LIN {X 0,Y 105.702,Z 1204.492,A -85,B 0,C 180,E1 2560.823,E2 2560.823} C_VEL
LIN {X 0,Y 120.882,Z 1198.363,A -85,B 0,C 180,E1 2552.47,E2 2552.47} C_VEL
LIN {X 0,Y 137.979,Z 1190.359,A -85,B 0,C 180,E1 2546.031,E2 2546.031} C_VEL
LIN {X 0,Y 156.407,Z 1180.629,A -85,B 0,C 180,E1 2541.04,E2 2541.04} C_VEL
LIN {X 0,Y 173.081,Z 1170.511,A -85,B 0,C 180,E1 2537.603,E2 2537.603} C_VEL
LIN {X 0,Y 192.101,Z 1157.421,A -85,B 0,C 180,E1 2534.511,E2 2534.511} C_VEL
LIN {X 0,Y 207.848,Z 1145.066,A -85,B 0,C 180,E1 2532.437,E2 2532.437} C_VEL
LIN {X 0,Y 225.86,Z 1129.001,A -85,B 0,C 180,E1 2530.458,E2 2530.458} C_VEL
LIN {X 0,Y 241.449,Z 1113.168,A -85,B 0,C 180,E1 2529.016,E2 2529.016} C_VEL
LIN {X 0,Y 256.349,Z 1095.766,A -85,B 0,C 180,E1 2527.823,E2 2527.823} C_VEL
LIN {X 0,Y 270.386,Z 1077.144,A -85,B 0,C 180,E1 2526.842,E2 2526.842} C_VEL
LIN {X 0,Y 283.038,Z 1057.453,A -85,B 0,C 180,E1 2526.055,E2 2526.055} C_VEL
LIN {X 0,Y 294.767,Z 1036.226,A -85,B 0,C 180,E1 2525.403,E2 2525.403} C_VEL
LIN {X 0,Y 304.085,Z 1016.178,A -85,B 0,C 180,E1 2524.939,E2 2524.939} C_VEL
LIN {X 0,Y 312.937,Z 993.046,A -85,B 0,C 180,E1 2524.54,E2 2524.54} C_VEL
LIN {X 0,Y 319.741,Z 970.772,A -85,B 0,C 180,E1 2524.255,E2 2524.255} C_VEL
LIN {X 0,Y 324.96,Z 947.508,A -85,B 0,C 180,E1 2523.991,E2 2523.991} C_VEL
LIN {X 0,Y 328.847,Z 922.27,A -85,B 0,C 180,E1 2523.717,E2 2523.717} C_VEL
LIN {X 0,Y 337.296,Z 853.105,A -85,B 0,C 180,E1 2522.984,E2 2522.984} C_VEL
LIN {X 0,Y 326.597,Z 938.266,A -85,B 0,C 180,E1 2522.039,E2 2522.039} C_VEL
LIN {X 0,Y 321.884,Z 961.652,A -85,B 0,C 180,E1 2521.748,E2 2521.748} C_VEL
LIN {X 0,Y 315.799,Z 984.104,A -85,B 0,C 180,E1 2521.402,E2 2521.402} C_VEL
LIN {X 0,Y 307.999,Z 1006.102,A -85,B 0,C 180,E1 2520.96,E2 2520.96} C_VEL
LIN {X 0,Y 298.407,Z 1028.316,A -85,B 0,C 180,E1 2520.384,E2 2520.384} C_VEL
LIN {X 0,Y 288.461,Z 1047.548,A -85,B 0,C 180,E1 2519.758,E2 2519.758} C_VEL
LIN {X 0,Y 275.512,Z 1068.916,A -85,B 0,C 180,E1 2518.888,E2 2518.888} C_VEL
LIN {X 0,Y 262.518,Z 1087.397,A -85,B 0,C 180,E1 2517.935,E2 2517.935} C_VEL
LIN {X 0,Y 247.376,Z 1106.017,A -85,B 0,C 180,E1 2516.694,E2 2516.694} C_VEL
LIN {X 0,Y 231.767,Z 1122.947,A -85,B 0,C 180,E1 2515.238,E2 2515.238} C_VEL
LIN {X 0,Y 215.365,Z 1138.404,A -85,B 0,C 180,E1 2513.473,E2 2513.473} C_VEL
LIN {X 0,Y 197.315,Z 1153.508,A -85,B 0,C 180,E1 2511.16,E2 2511.16} C_VEL
LIN {X 0,Y 179.971,Z 1166.226,A -85,B 0,C 180,E1 2508.462,E2 2508.462} C_VEL
LIN {X 0,Y 175.041,Z 1169.634,A -85,B 0,C 180,E1 2507.581,E2 2507.581} C_VEL
LIN {X 0,Y 168.74,Z 1173.521,A -85,B 0,C 180,E1 2506.765,E2 2506.765} C_VEL
LIN {X 0,Y 150.312,Z 1183.482,A -85,B 0,C 180,E1 2505.451,E2 2505.451} C_VEL
LIN {X 0,Y 144.844,Z 1186.245,A -85,B 0,C 180,E1 2504.485,E2 2504.485} C_VEL
LIN {X 0,Y 126.307,Z 1195.602,A -85,B 0,C 180,E1 2499.083,E2 2499.083} C_VEL
LIN {X 0,Y 108.864,Z 1203.189,A -85,B 0,C 180,E1 2491.849,E2 2491.849} C_VEL
LIN {X 0,Y 93.007,Z 1209.46,A -85,B 0,C 180,E1 2481.7,E2 2481.7} C_VEL
LIN {X 0,Y 81.228,Z 1213.752,A -85,B 0,C 180,E1 2468.886,E2 2468.886} C_VEL
LIN {X 0,Y 73.84,Z 1216.677,A -85,B 0,C 180,E1 2452.281,E2 2452.281} C_VEL
LIN {X 0,Y 72.017,Z 1217.75,A -85,B 0,C 180,E1 2437.98,E2 2437.98} C_VEL
LIN {X 0,Y 72.03,Z 1217.944,A -85,B 0,C 180,E1 2428.409,E2 2428.409} C_VEL
LIN {X 0,Y 72.337,Z 1217.462,A -85,B 0,C 180,E1 2416.41,E2 2416.41} C_VEL
LIN {X 0,Y 76.053,Z 1215.666,A -85,B 0,C 180,E1 2400.894,E2 2400.894} C_VEL
LIN {X 0,Y 85.042,Z 1212.358,A -85,B 0,C 180,E1 2386.078,E2 2386.078} C_VEL
LIN {X 0,Y 98.855,Z 1207.101,A -85,B 0,C 180,E1 2373.965,E2 2373.965} C_VEL
LIN {X 0,Y 115.778,Z 1200.203,A -85,B 0,C 180,E1 2364.936,E2 2364.936} C_VEL
LIN {X 0,Y 133.031,Z 1192.152,A -85,B 0,C 180,E1 2358.736,E2 2358.736} C_VEL
LIN {X 0,Y 152.349,Z 1181.996,A -85,B 0,C 180,E1 2353.757,E2 2353.757} C_VEL
LIN {X 0,Y 169.742,Z 1171.523,A -85,B 0,C 180,E1 2350.358,E2 2350.358} C_VEL
LIN {X 0,Y 189.984,Z 1157.647,A -85,B 0,C 180,E1 2347.257,E2 2347.257} C_VEL
LIN {X 0,Y 207.781,Z 1143.722,A -85,B 0,C 180,E1 2345.065,E2 2345.065} C_VEL
LIN {X 0,Y 225.332,Z 1127.955,A -85,B 0,C 180,E1 2343.257,E2 2343.257} C_VEL
LIN {X 0,Y 241.589,Z 1111.448,A -85,B 0,C 180,E1 2341.832,E2 2341.832} C_VEL
LIN {X 0,Y 256.663,Z 1093.76,A -85,B 0,C 180,E1 2340.67,E2 2340.67} C_VEL
LIN {X 0,Y 271.466,Z 1073.856,A -85,B 0,C 180,E1 2339.652,E2 2339.652} C_VEL
LIN {X 0,Y 283.511,Z 1055.087,A -85,B 0,C 180,E1 2338.901,E2 2338.901} C_VEL
LIN {X 0,Y 295.099,Z 1033.92,A -85,B 0,C 180,E1 2338.225,E2 2338.225} C_VEL
LIN {X 0,Y 304.701,Z 1013.197,A -85,B 0,C 180,E1 2337.702,E2 2337.702} C_VEL
LIN {X 0,Y 312.808,Z 991.691,A -85,B 0,C 180,E1 2337.278,E2 2337.278} C_VEL
LIN {X 0,Y 317.419,Z 977.052,A -85,B 0,C 180,E1 2337.025,E2 2337.025} C_VEL
LIN {X 0,Y 309.956,Z 999.939,A -85,B 0,C 180,E1 2336.744,E2 2336.744} C_VEL
LIN {X 0,Y 301.552,Z 1020.488,A -85,B 0,C 180,E1 2336.4,E2 2336.4} C_VEL
LIN {X 0,Y 290.701,Z 1042.634,A -85,B 0,C 180,E1 2335.902,E2 2335.902} C_VEL
LIN {X 0,Y 279.88,Z 1061.31,A -85,B 0,C 180,E1 2335.352,E2 2335.352} C_VEL
LIN {X 0,Y 266.156,Z 1081.659,A -85,B 0,C 180,E1 2334.57,E2 2334.57} C_VEL
LIN {X 0,Y 252.01,Z 1099.859,A -85,B 0,C 180,E1 2333.65,E2 2333.65} C_VEL
LIN {X 0,Y 236.489,Z 1117.088,A -85,B 0,C 180,E1 2332.5,E2 2332.5} C_VEL
LIN {X 0,Y 220.612,Z 1132.702,A -85,B 0,C 180,E1 2331.121,E2 2331.121} C_VEL
LIN {X 0,Y 203.466,Z 1147.304,A -85,B 0,C 180,E1 2329.365,E2 2329.365} C_VEL
LIN {X 0,Y 184.695,Z 1161.384,A -85,B 0,C 180,E1 2327.018,E2 2327.018} C_VEL
LIN {X 0,Y 167.217,Z 1172.785,A -85,B 0,C 180,E1 2324.298,E2 2324.298} C_VEL
LIN {X 0,Y 147.575,Z 1183.95,A -85,B 0,C 180,E1 2320.349,E2 2320.349} C_VEL
LIN {X 0,Y 129.663,Z 1192.8,A -85,B 0,C 180,E1 2315.494,E2 2315.494} C_VEL
LIN {X 0,Y 111.422,Z 1200.526,A -85,B 0,C 180,E1 2308.484,E2 2308.484} C_VEL
LIN {X 0,Y 95.371,Z 1206.516,A -85,B 0,C 180,E1 2299.011,E2 2299.011} C_VEL
LIN {X 0,Y 83.103,Z 1210.53,A -85,B 0,C 180,E1 2286.983,E2 2286.983} C_VEL
LIN {X 0,Y 74.655,Z 1213.263,A -85,B 0,C 180,E1 2270.357,E2 2270.357} C_VEL
LIN {X 0,Y 72.2,Z 1214.155,A -85,B 0,C 180,E1 2255.563,E2 2255.563} C_VEL
LIN {X 0,Y 72.16,Z 1214.185,A -85,B 0,C 180,E1 2245.231,E2 2245.231} C_VEL
LIN {X 0,Y 74,Z 1213.483,A -85,B 0,C 180,E1 2231.895,E2 2231.895} C_VEL
LIN {X 0,Y 80.832,Z 1211.371,A -85,B 0,C 180,E1 2216.177,E2 2216.177} C_VEL
LIN {X 0,Y 92.82,Z 1207.406,A -85,B 0,C 180,E1 2202.904,E2 2202.904} C_VEL
LIN {X 0,Y 109.122,Z 1201.539,A -85,B 0,C 180,E1 2192.545,E2 2192.545} C_VEL
LIN {X 0,Y 125.492,Z 1194.778,A -85,B 0,C 180,E1 2185.799,E2 2185.799} C_VEL
LIN {X 0,Y 144.029,Z 1185.943,A -85,B 0,C 180,E1 2180.417,E2 2180.417} C_VEL
LIN {X 0,Y 161.73,Z 1176.279,A -85,B 0,C 180,E1 2176.615,E2 2176.615} C_VEL
LIN {X 0,Y 180.001,Z 1164.784,A -85,B 0,C 180,E1 2173.572,E2 2173.572} C_VEL
LIN {X 0,Y 197.751,Z 1152.12,A -85,B 0,C 180,E1 2171.22,E2 2171.22} C_VEL
LIN {X 0,Y 214.827,Z 1138.084,A -85,B 0,C 180,E1 2169.357,E2 2169.357} C_VEL
LIN {X 0,Y 231.141,Z 1122.991,A -85,B 0,C 180,E1 2167.865,E2 2167.865} C_VEL
LIN {X 0,Y 246.625,Z 1106.46,A -85,B 0,C 180,E1 2166.652,E2 2166.652} C_VEL
LIN {X 0,Y 261.237,Z 1088.836,A -85,B 0,C 180,E1 2165.662,E2 2165.662} C_VEL
LIN {X 0,Y 274.451,Z 1070.287,A -85,B 0,C 180,E1 2164.87,E2 2164.87} C_VEL
LIN {X 0,Y 287.221,Z 1049.628,A -85,B 0,C 180,E1 2164.192,E2 2164.192} C_VEL
LIN {X 0,Y 297.576,Z 1029.866,A -85,B 0,C 180,E1 2163.697,E2 2163.697} C_VEL
LIN {X 0,Y 307.457,Z 1007.353,A -85,B 0,C 180,E1 2163.274,E2 2163.274} C_VEL
LIN {X 0,Y 315.059,Z 986.183,A -85,B 0,C 180,E1 2162.986,E2 2162.986} C_VEL
LIN {X 0,Y 316.8,Z 980.517,A -85,B 0,C 180,E1 2162.918,E2 2162.918} C_VEL
LIN {X 0,Y 308.808,Z 1003.784,A -85,B 0,C 180,E1 2162.503,E2 2162.503} C_VEL
LIN {X 0,Y 300.145,Z 1024.367,A -85,B 0,C 180,E1 2162.032,E2 2162.032} C_VEL
LIN {X 0,Y 289.549,Z 1045.161,A -85,B 0,C 180,E1 2161.44,E2 2161.44} C_VEL
LIN {X 0,Y 277.655,Z 1065.235,A -85,B 0,C 180,E1 2160.725,E2 2160.725} C_VEL
LIN {X 0,Y 264.462,Z 1084.134,A -85,B 0,C 180,E1 2159.872,E2 2159.872} C_VEL
LIN {X 0,Y 249.52,Z 1102.865,A -85,B 0,C 180,E1 2158.787,E2 2158.787} C_VEL
LIN {X 0,Y 234.183,Z 1119.573,A -85,B 0,C 180,E1 2157.535,E2 2157.535} C_VEL
LIN {X 0,Y 216.533,Z 1136.41,A -85,B 0,C 180,E1 2155.863,E2 2155.863} C_VEL
LIN {X 0,Y 199.097,Z 1151.041,A -85,B 0,C 180,E1 2153.905,E2 2153.905} C_VEL
LIN {X 0,Y 180.729,Z 1164.455,A -85,B 0,C 180,E1 2151.409,E2 2151.409} C_VEL
LIN {X 0,Y 162.233,Z 1176.458,A -85,B 0,C 180,E1 2148.265,E2 2148.265} C_VEL
LIN {X 0,Y 144.844,Z 1186.245,A -85,B 0,C 180,E1 2144.485,E2 2144.485} C_VEL
LIN {X 0,Y 138.393,Z 1189.511,A -85,B 0,C 180,E1 2143.29,E2 2143.29} C_VEL
LIN {X 0,Y 120.351,Z 1196.925,A -85,B 0,C 180,E1 2141.09,E2 2141.09} C_VEL
LIN {X 0,Y 113.904,Z 1199.508,A -85,B 0,C 180,E1 2139.414,E2 2139.414} C_VEL
LIN {X 0,Y 95.954,Z 1206.45,A -85,B 0,C 180,E1 2131.08,E2 2131.08} C_VEL
LIN {X 0,Y 81.07,Z 1211.613,A -85,B 0,C 180,E1 2119.877,E2 2119.877} C_VEL
LIN {X 0,Y 69.737,Z 1215.254,A -85,B 0,C 180,E1 2103.998,E2 2103.998} C_VEL
LIN {X 0,Y 64.714,Z 1217.132,A -85,B 0,C 180,E1 2087.071,E2 2087.071} C_VEL
LIN {X 0,Y 64.013,Z 1217.723,A -85,B 0,C 180,E1 2072.686,E2 2072.686} C_VEL
LIN {X 0,Y 64.003,Z 1217.615,A -85,B 0,C 180,E1 2063.722,E2 2063.722} C_VEL
LIN {X 0,Y 65.464,Z 1216.757,A -85,B 0,C 180,E1 2048.703,E2 2048.703} C_VEL
LIN {X 0,Y 72.619,Z 1214.323,A -85,B 0,C 180,E1 2030.702,E2 2030.702} C_VEL
LIN {X 0,Y 84.806,Z 1210.252,A -85,B 0,C 180,E1 2016.706,E2 2016.706} C_VEL
LIN {X 0,Y 101.269,Z 1204.428,A -85,B 0,C 180,E1 2006.043,E2 2006.043} C_VEL
LIN {X 0,Y 118.415,Z 1197.441,A -85,B 0,C 180,E1 1998.97,E2 1998.97} C_VEL
LIN {X 0,Y 138.672,Z 1188.015,A -85,B 0,C 180,E1 1993.251,E2 1993.251} C_VEL
LIN {X 0,Y 157.115,Z 1178.086,A -85,B 0,C 180,E1 1989.461,E2 1989.461} C_VEL
LIN {X 0,Y 177.052,Z 1165.75,A -85,B 0,C 180,E1 1986.324,E2 1986.324} C_VEL
LIN {X 0,Y 195.455,Z 1152.75,A -85,B 0,C 180,E1 1984.031,E2 1984.031} C_VEL
LIN {X 0,Y 213.903,Z 1137.723,A -85,B 0,C 180,E1 1982.143,E2 1982.143} C_VEL
LIN {X 0,Y 231.481,Z 1121.442,A -85,B 0,C 180,E1 1980.634,E2 1980.634} C_VEL
LIN {X 0,Y 246.974,Z 1104.919,A -85,B 0,C 180,E1 1979.483,E2 1979.483} C_VEL
LIN {X 0,Y 263.061,Z 1085.24,A -85,B 0,C 180,E1 1978.43,E2 1978.43} C_VEL
LIN {X 0,Y 276.189,Z 1066.705,A -85,B 0,C 180,E1 1977.666,E2 1977.666} C_VEL
LIN {X 0,Y 284.295,Z 1053.752,A -85,B 0,C 180,E1 1977.214,E2 1977.214} C_VEL
LIN {X 0,Y 271.987,Z 1072.972,A -85,B 0,C 180,E1 1976.628,E2 1976.628} C_VEL
LIN {X 0,Y 256.654,Z 1093.584,A -85,B 0,C 180,E1 1975.794,E2 1975.794} C_VEL
LIN {X 0,Y 241.933,Z 1110.756,A -85,B 0,C 180,E1 1974.874,E2 1974.874} C_VEL
LIN {X 0,Y 225.34,Z 1127.498,A -85,B 0,C 180,E1 1973.674,E2 1973.674} C_VEL
LIN {X 0,Y 207.908,Z 1142.981,A -85,B 0,C 180,E1 1972.172,E2 1972.172} C_VEL
LIN {X 0,Y 190.648,Z 1156.247,A -85,B 0,C 180,E1 1970.391,E2 1970.391} C_VEL
LIN {X 0,Y 171.743,Z 1169.043,A -85,B 0,C 180,E1 1967.977,E2 1967.977} C_VEL
LIN {X 0,Y 153.222,Z 1179.86,A -85,B 0,C 180,E1 1964.968,E2 1964.968} C_VEL
LIN {X 0,Y 132.596,Z 1190.229,A -85,B 0,C 180,E1 1960.489,E2 1960.489} C_VEL
LIN {X 0,Y 113.874,Z 1198.315,A -85,B 0,C 180,E1 1954.74,E2 1954.74} C_VEL
LIN {X 0,Y 95.933,Z 1204.811,A -85,B 0,C 180,E1 1946.49,E2 1946.49} C_VEL
LIN {X 0,Y 80.678,Z 1209.653,A -85,B 0,C 180,E1 1934.944,E2 1934.944} C_VEL
LIN {X 0,Y 70.026,Z 1212.639,A -85,B 0,C 180,E1 1919.983,E2 1919.983} C_VEL
LIN {X 0,Y 64.708,Z 1214.235,A -85,B 0,C 180,E1 1901.588,E2 1901.588} C_VEL
LIN {X 0,Y 64.092,Z 1214.476,A -85,B 0,C 180,E1 1888.212,E2 1888.212} C_VEL
LIN {X 0,Y 65.755,Z 1213.882,A -85,B 0,C 180,E1 1872.295,E2 1872.295} C_VEL
LIN {X 0,Y 71.984,Z 1212.139,A -85,B 0,C 180,E1 1856.248,E2 1856.248} C_VEL
LIN {X 0,Y 84.9,Z 1208.419,A -85,B 0,C 180,E1 1841.086,E2 1841.086} C_VEL
LIN {X 0,Y 100.349,Z 1203.42,A -85,B 0,C 180,E1 1831.032,E2 1831.032} C_VEL
LIN {X 0,Y 118.798,Z 1196.378,A -85,B 0,C 180,E1 1823.453,E2 1823.453} C_VEL
LIN {X 0,Y 137.838,Z 1187.977,A -85,B 0,C 180,E1 1818.148,E2 1818.148} C_VEL
LIN {X 0,Y 156.838,Z 1178.026,A -85,B 0,C 180,E1 1814.301,E2 1814.301} C_VEL
LIN {X 0,Y 176.392,Z 1166.281,A -85,B 0,C 180,E1 1811.296,E2 1811.296} C_VEL
LIN {X 0,Y 193.469,Z 1154.447,A -85,B 0,C 180,E1 1809.215,E2 1809.215} C_VEL
LIN {X 0,Y 213.018,Z 1138.919,A -85,B 0,C 180,E1 1807.281,E2 1807.281} C_VEL
LIN {X 0,Y 229.203,Z 1124.197,A -85,B 0,C 180,E1 1805.953,E2 1805.953} C_VEL
LIN {X 0,Y 245.334,Z 1107.345,A -85,B 0,C 180,E1 1804.824,E2 1804.824} C_VEL
LIN {X 0,Y 260.076,Z 1089.844,A -85,B 0,C 180,E1 1803.936,E2 1803.936} C_VEL
LIN {X 0,Y 273.888,Z 1070.725,A -85,B 0,C 180,E1 1803.202,E2 1803.202} C_VEL
LIN {X 0,Y 283.669,Z 1055.389,A -85,B 0,C 180,E1 1802.726,E2 1802.726} C_VEL
LIN {X 0,Y 271.636,Z 1073.968,A -85,B 0,C 180,E1 1802.059,E2 1802.059} C_VEL
LIN {X 0,Y 257.016,Z 1093.457,A -85,B 0,C 180,E1 1801.169,E2 1801.169} C_VEL
LIN {X 0,Y 241.966,Z 1110.953,A -85,B 0,C 180,E1 1800.143,E2 1800.143} C_VEL
LIN {X 0,Y 226.008,Z 1127.059,A -85,B 0,C 180,E1 1798.91,E2 1798.91} C_VEL
LIN {X 0,Y 208.202,Z 1142.955,A -85,B 0,C 180,E1 1797.296,E2 1797.296} C_VEL
LIN {X 0,Y 189.615,Z 1157.281,A -85,B 0,C 180,E1 1795.281,E2 1795.281} C_VEL
LIN {X 0,Y 169.254,Z 1170.994,A -85,B 0,C 180,E1 1792.532,E2 1792.532} C_VEL
LIN {X 0,Y 150.463,Z 1182.017,A -85,B 0,C 180,E1 1789.276,E2 1789.276} C_VEL
LIN {X 0,Y 130.605,Z 1192.072,A -85,B 0,C 180,E1 1784.71,E2 1784.71} C_VEL
LIN {X 0,Y 113.904,Z 1199.508,A -85,B 0,C 180,E1 1779.414,E2 1779.414} C_VEL
LIN {X 0,Y 107.512,Z 1201.995,A -85,B 0,C 180,E1 1777.527,E2 1777.527} C_VEL
LIN {X 0,Y 88.575,Z 1207.694,A -85,B 0,C 180,E1 1772.939,E2 1772.939} C_VEL
LIN {X 0,Y 83.353,Z 1209.156,A -85,B 0,C 180,E1 1770.348,E2 1770.348} C_VEL
LIN {X 0,Y 69.186,Z 1213.331,A -85,B 0,C 180,E1 1757.48,E2 1757.48} C_VEL
LIN {X 0,Y 59.062,Z 1216.261,A -85,B 0,C 180,E1 1738.295,E2 1738.295} C_VEL
LIN {X 0,Y 56.045,Z 1217.365,A -85,B 0,C 180,E1 1719.239,E2 1719.239} C_VEL
LIN {X 0,Y 56.025,Z 1217.538,A -85,B 0,C 180,E1 1708.084,E2 1708.084} C_VEL
LIN {X 0,Y 56.841,Z 1216.973,A -85,B 0,C 180,E1 1691.541,E2 1691.541} C_VEL
LIN {X 0,Y 62.669,Z 1215.125,A -85,B 0,C 180,E1 1672.68,E2 1672.68} C_VEL
LIN {X 0,Y 75.344,Z 1211.544,A -85,B 0,C 180,E1 1655.953,E2 1655.953} C_VEL
LIN {X 0,Y 91.433,Z 1206.409,A -85,B 0,C 180,E1 1644.819,E2 1644.819} C_VEL
LIN {X 0,Y 110.686,Z 1199.399,A -85,B 0,C 180,E1 1636.759,E2 1636.759} C_VEL
LIN {X 0,Y 129.581,Z 1191.294,A -85,B 0,C 180,E1 1631.496,E2 1631.496} C_VEL
LIN {X 0,Y 151.275,Z 1180.431,A -85,B 0,C 180,E1 1627.215,E2 1627.215} C_VEL
LIN {X 0,Y 171.448,Z 1168.708,A -85,B 0,C 180,E1 1624.258,E2 1624.258} C_VEL
LIN {X 0,Y 191.089,Z 1155.345,A -85,B 0,C 180,E1 1622.001,E2 1622.001} C_VEL
LIN {X 0,Y 209.972,Z 1140.676,A -85,B 0,C 180,E1 1620.246,E2 1620.246} C_VEL
LIN {X 0,Y 227.008,Z 1125.474,A -85,B 0,C 180,E1 1618.914,E2 1618.914} C_VEL
LIN {X 0,Y 244.15,Z 1107.94,A -85,B 0,C 180,E1 1617.766,E2 1617.766} C_VEL
LIN {X 0,Y 251.238,Z 1099.995,A -85,B 0,C 180,E1 1617.323,E2 1617.323} C_VEL
LIN {X 0,Y 235.425,Z 1117.216,A -85,B 0,C 180,E1 1616.421,E2 1616.421} C_VEL
LIN {X 0,Y 218.411,Z 1133.512,A -85,B 0,C 180,E1 1615.273,E2 1615.273} C_VEL
LIN {X 0,Y 201.114,Z 1147.828,A -85,B 0,C 180,E1 1613.889,E2 1613.889} C_VEL
LIN {X 0,Y 181.747,Z 1161.863,A -85,B 0,C 180,E1 1611.991,E2 1611.991} C_VEL
LIN {X 0,Y 163.579,Z 1173.248,A -85,B 0,C 180,E1 1609.766,E2 1609.766} C_VEL
LIN {X 0,Y 142.938,Z 1184.39,A -85,B 0,C 180,E1 1606.485,E2 1606.485} C_VEL
LIN {X 0,Y 123.815,Z 1193.239,A -85,B 0,C 180,E1 1602.345,E2 1602.345} C_VEL
LIN {X 0,Y 103.902,Z 1200.933,A -85,B 0,C 180,E1 1596.16,E2 1596.16} C_VEL
LIN {X 0,Y 85.606,Z 1206.932,A -85,B 0,C 180,E1 1587.239,E2 1587.239} C_VEL
LIN {X 0,Y 70.837,Z 1210.947,A -85,B 0,C 180,E1 1574.89,E2 1574.89} C_VEL
LIN {X 0,Y 59.805,Z 1213.672,A -85,B 0,C 180,E1 1555.765,E2 1555.765} C_VEL
LIN {X 0,Y 56.272,Z 1214.564,A -85,B 0,C 180,E1 1537.145,E2 1537.145} C_VEL
LIN {X 0,Y 56.168,Z 1214.615,A -85,B 0,C 180,E1 1524.894,E2 1524.894} C_VEL
LIN {X 0,Y 58.901,Z 1213.893,A -85,B 0,C 180,E1 1507.019,E2 1507.019} C_VEL
LIN {X 0,Y 68.522,Z 1211.632,A -85,B 0,C 180,E1 1487.839,E2 1487.839} C_VEL
LIN {X 0,Y 82.63,Z 1207.82,A -85,B 0,C 180,E1 1474.632,E2 1474.632} C_VEL
LIN {X 0,Y 101.313,Z 1201.963,A -85,B 0,C 180,E1 1464.777,E2 1464.777} C_VEL
LIN {X 0,Y 119.322,Z 1195.2,A -85,B 0,C 180,E1 1458.759,E2 1458.759} C_VEL
LIN {X 0,Y 140.122,Z 1185.931,A -85,B 0,C 180,E1 1453.966,E2 1453.966} C_VEL
LIN {X 0,Y 159.752,Z 1175.708,A -85,B 0,C 180,E1 1450.694,E2 1450.694} C_VEL
LIN {X 0,Y 178.826,Z 1164.005,A -85,B 0,C 180,E1 1448.253,E2 1448.253} C_VEL
LIN {X 0,Y 197.196,Z 1151.194,A -85,B 0,C 180,E1 1446.388,E2 1446.388} C_VEL
LIN {X 0,Y 214.76,Z 1136.954,A -85,B 0,C 180,E1 1444.92,E2 1444.92} C_VEL
LIN {X 0,Y 232.449,Z 1120.635,A -85,B 0,C 180,E1 1443.691,E2 1443.691} C_VEL
LIN {X 0,Y 247.262,Z 1104.924,A -85,B 0,C 180,E1 1442.815,E2 1442.815} C_VEL
LIN {X 0,Y 250.75,Z 1101.032,A -85,B 0,C 180,E1 1442.613,E2 1442.613} C_VEL
LIN {X 0,Y 234.796,Z 1118.183,A -85,B 0,C 180,E1 1441.611,E2 1441.611} C_VEL
LIN {X 0,Y 216.972,Z 1134.999,A -85,B 0,C 180,E1 1440.309,E2 1440.309} C_VEL
LIN {X 0,Y 200.008,Z 1148.95,A -85,B 0,C 180,E1 1438.854,E2 1438.854} C_VEL
LIN {X 0,Y 180.254,Z 1163.149,A -85,B 0,C 180,E1 1436.803,E2 1436.803} C_VEL
LIN {X 0,Y 160.781,Z 1175.334,A -85,B 0,C 180,E1 1434.266,E2 1434.266} C_VEL
LIN {X 0,Y 140.759,Z 1186.074,A -85,B 0,C 180,E1 1430.882,E2 1430.882} C_VEL
LIN {X 0,Y 120.469,Z 1195.536,A -85,B 0,C 180,E1 1426.184,E2 1426.184} C_VEL
LIN {X 0,Y 101.245,Z 1203.068,A -85,B 0,C 180,E1 1419.749,E2 1419.749} C_VEL
LIN {X 0,Y 83.353,Z 1209.156,A -85,B 0,C 180,E1 1410.348,E2 1410.348} C_VEL
LIN {X 0,Y 77.397,Z 1210.761,A -85,B 0,C 180,E1 1406.968,E2 1406.968} C_VEL
LIN {X 0,Y 59.712,Z 1214.327,A -85,B 0,C 180,E1 1396.599,E2 1396.599} C_VEL
LIN {X 0,Y 56.049,Z 1215.032,A -85,B 0,C 180,E1 1391.802,E2 1391.802} C_VEL
LIN {X 0,Y 48.839,Z 1216.936,A -85,B 0,C 180,E1 1369.12,E2 1369.12} C_VEL
LIN {X 0,Y 48.037,Z 1217.362,A -85,B 0,C 180,E1 1351.193,E2 1351.193} C_VEL
LIN {X 0,Y 48.237,Z 1217.098,A -85,B 0,C 180,E1 1336.82,E2 1336.82} C_VEL
LIN {X 0,Y 54.007,Z 1215.516,A -85,B 0,C 180,E1 1312.342,E2 1312.342} C_VEL
LIN {X 0,Y 65.891,Z 1212.561,A -85,B 0,C 180,E1 1294.974,E2 1294.974} C_VEL
LIN {X 0,Y 84.096,Z 1207.511,A -85,B 0,C 180,E1 1281.971,E2 1281.971} C_VEL
LIN {X 0,Y 102.245,Z 1201.497,A -85,B 0,C 180,E1 1274.506,E2 1274.506} C_VEL
LIN {X 0,Y 123.45,Z 1193.147,A -85,B 0,C 180,E1 1268.844,E2 1268.844} C_VEL
LIN {X 0,Y 143.552,Z 1183.812,A -85,B 0,C 180,E1 1265.12,E2 1265.12} C_VEL
LIN {X 0,Y 164.107,Z 1172.563,A -85,B 0,C 180,E1 1262.283,E2 1262.283} C_VEL
LIN {X 0,Y 183.974,Z 1160.06,A -85,B 0,C 180,E1 1260.166,E2 1260.166} C_VEL
LIN {X 0,Y 203.038,Z 1146.049,A -85,B 0,C 180,E1 1258.525,E2 1258.525} C_VEL
LIN {X 0,Y 218.391,Z 1133.367,A -85,B 0,C 180,E1 1257.421,E2 1257.421} C_VEL
LIN {X 0,Y 200.416,Z 1148.093,A -85,B 0,C 180,E1 1256.183,E2 1256.183} C_VEL
LIN {X 0,Y 180.798,Z 1162.106,A -85,B 0,C 180,E1 1254.529,E2 1254.529} C_VEL
LIN {X 0,Y 162.19,Z 1173.568,A -85,B 0,C 180,E1 1252.561,E2 1252.561} C_VEL
LIN {X 0,Y 141.264,Z 1184.61,A -85,B 0,C 180,E1 1249.683,E2 1249.683} C_VEL
LIN {X 0,Y 121.6,Z 1193.458,A -85,B 0,C 180,E1 1245.991,E2 1245.991} C_VEL
LIN {X 0,Y 101.728,Z 1200.86,A -85,B 0,C 180,E1 1240.657,E2 1240.657} C_VEL
LIN {X 0,Y 82.3,Z 1206.938,A -85,B 0,C 180,E1 1232.483,E2 1232.483} C_VEL
LIN {X 0,Y 65.348,Z 1211.155,A -85,B 0,C 180,E1 1219.909,E2 1219.909} C_VEL
LIN {X 0,Y 52.656,Z 1213.878,A -85,B 0,C 180,E1 1199.584,E2 1199.584} C_VEL
LIN {X 0,Y 48.331,Z 1214.769,A -85,B 0,C 180,E1 1178.327,E2 1178.327} C_VEL
LIN {X 0,Y 48.196,Z 1214.82,A -85,B 0,C 180,E1 1164.046,E2 1164.046} C_VEL
LIN {X 0,Y 51.572,Z 1214.099,A -85,B 0,C 180,E1 1143.518,E2 1143.518} C_VEL
LIN {X 0,Y 62.754,Z 1211.84,A -85,B 0,C 180,E1 1122.868,E2 1122.868} C_VEL
LIN {X 0,Y 78.304,Z 1208.03,A -85,B 0,C 180,E1 1109.74,E2 1109.74} C_VEL
LIN {X 0,Y 98.187,Z 1202.175,A -85,B 0,C 180,E1 1100.47,E2 1100.47} C_VEL
LIN {X 0,Y 116.964,Z 1195.414,A -85,B 0,C 180,E1 1094.991,E2 1094.991} C_VEL
LIN {X 0,Y 138.389,Z 1186.152,A -85,B 0,C 180,E1 1090.705,E2 1090.705} C_VEL
LIN {X 0,Y 158.449,Z 1175.93,A -85,B 0,C 180,E1 1087.815,E2 1087.815} C_VEL
LIN {X 0,Y 177.845,Z 1164.244,A -85,B 0,C 180,E1 1085.673,E2 1085.673} C_VEL
LIN {X 0,Y 196.462,Z 1151.451,A -85,B 0,C 180,E1 1084.048,E2 1084.048} C_VEL
LIN {X 0,Y 214.22,Z 1137.228,A -85,B 0,C 180,E1 1082.772,E2 1082.772} C_VEL
LIN {X 0,Y 217.794,Z 1134.195,A -85,B 0,C 180,E1 1082.526,E2 1082.526} C_VEL
LIN {X 0,Y 200.016,Z 1148.682,A -85,B 0,C 180,E1 1081.222,E2 1081.222} C_VEL
LIN {X 0,Y 179.227,Z 1163.398,A -85,B 0,C 180,E1 1079.361,E2 1079.361} C_VEL
LIN {X 0,Y 159.182,Z 1175.678,A -85,B 0,C 180,E1 1077.094,E2 1077.094} C_VEL
LIN {X 0,Y 138.719,Z 1186.321,A -85,B 0,C 180,E1 1074.084,E2 1074.084} C_VEL
LIN {X 0,Y 117.825,Z 1195.683,A -85,B 0,C 180,E1 1069.857,E2 1069.857} C_VEL
LIN {X 0,Y 97.795,Z 1203.167,A -85,B 0,C 180,E1 1063.956,E2 1063.956} C_VEL
LIN {X 0,Y 77.643,Z 1209.47,A -85,B 0,C 180,E1 1054.347,E2 1054.347} C_VEL
LIN {X 0,Y 62.629,Z 1213.454,A -85,B 0,C 180,E1 1041.469,E2 1041.469} C_VEL
LIN {X 0,Y 56.049,Z 1215.032,A -85,B 0,C 180,E1 1031.802,E2 1031.802} C_VEL
LIN {X 0,Y 51.852,Z 1215.904,A -85,B 0,C 180,E1 1024.917,E2 1024.917} C_VEL
LIN {X 0,Y 44.201,Z 1216.787,A -85,B 0,C 180,E1 1011.709,E2 1011.709} C_VEL
LIN {X 0,Y 40.097,Z 1217.089,A -85,B 0,C 180,E1 995.755,E2 995.755} C_VEL
LIN {X 0,Y 40.015,Z 1217.138,A -85,B 0,C 180,E1 992.54,E2 992.54} C_VEL
LIN {X 0,Y 40.122,Z 1216.971,A -85,B 0,C 180,E1 978.5,E2 978.5} C_VEL
LIN {X 0,Y 44.891,Z 1215.894,A -85,B 0,C 180,E1 953.032,E2 953.032} C_VEL
LIN {X 0,Y 58.575,Z 1213.02,A -85,B 0,C 180,E1 931.407,E2 931.407} C_VEL
LIN {X 0,Y 76.143,Z 1208.757,A -85,B 0,C 180,E1 919.011,E2 919.011} C_VEL
LIN {X 0,Y 96.759,Z 1202.531,A -85,B 0,C 180,E1 910.986,E2 910.986} C_VEL
LIN {X 0,Y 118.063,Z 1194.791,A -85,B 0,C 180,E1 905.833,E2 905.833} C_VEL
LIN {X 0,Y 139.096,Z 1185.462,A -85,B 0,C 180,E1 902.341,E2 902.341} C_VEL
LIN {X 0,Y 160.979,Z 1174.067,A -85,B 0,C 180,E1 899.697,E2 899.697} C_VEL
LIN {X 0,Y 180.093,Z 1162.426,A -85,B 0,C 180,E1 897.917,E2 897.917} C_VEL
LIN {X 0,Y 185.359,Z 1158.943,A -85,B 0,C 180,E1 897.49,E2 897.49} C_VEL
LIN {X 0,Y 165.418,Z 1171.447,A -85,B 0,C 180,E1 895.811,E2 895.811} C_VEL
LIN {X 0,Y 144.89,Z 1182.561,A -85,B 0,C 180,E1 893.571,E2 893.571} C_VEL
LIN {X 0,Y 124.652,Z 1191.679,A -85,B 0,C 180,E1 890.611,E2 890.611} C_VEL
LIN {X 0,Y 103.018,Z 1199.879,A -85,B 0,C 180,E1 886.064,E2 886.064} C_VEL
LIN {X 0,Y 83.132,Z 1205.957,A -85,B 0,C 180,E1 879.585,E2 879.585} C_VEL
LIN {X 0,Y 63.436,Z 1210.74,A -85,B 0,C 180,E1 868.335,E2 868.335} C_VEL
LIN {X 0,Y 48.808,Z 1213.589,A -85,B 0,C 180,E1 850.96,E2 850.96} C_VEL
LIN {X 0,Y 40.813,Z 1214.911,A -85,B 0,C 180,E1 824.181,E2 824.181} C_VEL
LIN {X 0,Y 40.137,Z 1215.067,A -85,B 0,C 180,E1 805.714,E2 805.714} C_VEL
LIN {X 0,Y 43.731,Z 1214.435,A -85,B 0,C 180,E1 781.306,E2 781.306} C_VEL
LIN {X 0,Y 54.828,Z 1212.539,A -85,B 0,C 180,E1 760.012,E2 760.012} C_VEL
LIN {X 0,Y 72.123,Z 1208.844,A -85,B 0,C 180,E1 745.696,E2 745.696} C_VEL
LIN {X 0,Y 92.033,Z 1203.546,A -85,B 0,C 180,E1 737.051,E2 737.051} C_VEL
LIN {X 0,Y 112.306,Z 1196.672,A -85,B 0,C 180,E1 731.672,E2 731.672} C_VEL
LIN {X 0,Y 133.256,Z 1188.187,A -85,B 0,C 180,E1 727.934,E2 727.934} C_VEL
LIN {X 0,Y 153.638,Z 1178.194,A -85,B 0,C 180,E1 725.314,E2 725.314} C_VEL
LIN {X 0,Y 175.254,Z 1165.741,A -85,B 0,C 180,E1 723.235,E2 723.235} C_VEL
LIN {X 0,Y 184.893,Z 1159.534,A -85,B 0,C 180,E1 722.46,E2 722.46} C_VEL
LIN {X 0,Y 164.895,Z 1172.004,A -85,B 0,C 180,E1 720.695,E2 720.695} C_VEL
LIN {X 0,Y 144.041,Z 1183.284,A -85,B 0,C 180,E1 718.314,E2 718.314} C_VEL
LIN {X 0,Y 123.421,Z 1192.659,A -85,B 0,C 180,E1 715.166,E2 715.166} C_VEL
LIN {X 0,Y 100.49,Z 1201.393,A -85,B 0,C 180,E1 710.075,E2 710.075} C_VEL
LIN {X 0,Y 80.484,Z 1207.649,A -85,B 0,C 180,E1 703.053,E2 703.053} C_VEL
LIN {X 0,Y 61.536,Z 1212.408,A -85,B 0,C 180,E1 691.33,E2 691.33} C_VEL
LIN {X 0,Y 47.264,Z 1215.468,A -85,B 0,C 180,E1 672.606,E2 672.606} C_VEL
LIN {X 0,Y 40.29,Z 1216.926,A -85,B 0,C 180,E1 644.369,E2 644.369} C_VEL
LIN {X 0,Y 40.015,Z 1217.138,A -85,B 0,C 180,E1 632.54,E2 632.54} C_VEL
LIN {X 0,Y 39.579,Z 1217.192,A -85,B 0,C 180,E1 623.87,E2 623.87} C_VEL
LIN {X 0,Y 38.17,Z 1216.998,A -85,B 0,C 180,E1 611.719,E2 611.719} C_VEL
LIN {X 0,Y 38.593,Z 1215.902,A -85,B 0,C 180,E1 587.69,E2 587.69} C_VEL
LIN {X 0,Y 41.205,Z 1215.294,A -85,B 0,C 180,E1 580.447,E2 580.447} C_VEL
LIN {X 0,Y 57.194,Z 1212.307,A -85,B 0,C 180,E1 562.098,E2 562.098} C_VEL
LIN {X 0,Y 77.541,Z 1207.604,A -85,B 0,C 180,E1 551.481,E2 551.481} C_VEL
LIN {X 0,Y 98.425,Z 1201.378,A -85,B 0,C 180,E1 545.414,E2 545.414} C_VEL
LIN {X 0,Y 122.005,Z 1192.698,A -85,B 0,C 180,E1 541.112,E2 541.112} C_VEL
LIN {X 0,Y 143.03,Z 1183.361,A -85,B 0,C 180,E1 538.482,E2 538.482} C_VEL
LIN {X 0,Y 152.119,Z 1178.733,A -85,B 0,C 180,E1 537.537,E2 537.537} C_VEL
LIN {X 0,Y 131.414,Z 1188.68,A -85,B 0,C 180,E1 535.346,E2 535.346} C_VEL
LIN {X 0,Y 109.752,Z 1197.184,A -85,B 0,C 180,E1 532.145,E2 532.145} C_VEL
LIN {X 0,Y 87.207,Z 1204.402,A -85,B 0,C 180,E1 527.047,E2 527.047} C_VEL
LIN {X 0,Y 67.268,Z 1209.373,A -85,B 0,C 180,E1 519.457,E2 519.457} C_VEL
LIN {X 0,Y 47.826,Z 1213.028,A -85,B 0,C 180,E1 504.621,E2 504.621} C_VEL
LIN {X 0,Y 35.58,Z 1214.808,A -85,B 0,C 180,E1 480.387,E2 480.387} C_VEL
LIN {X 0,Y 32.1,Z 1215.326,A -85,B 0,C 180,E1 450,E2 450} C_VEL
LIN {X 0,Y 35.563,Z 1214.835,A -85,B 0,C 180,E1 419.597,E2 419.597} C_VEL
LIN {X 0,Y 47.797,Z 1213.075,A -85,B 0,C 180,E1 395.331,E2 395.331} C_VEL
LIN {X 0,Y 67.239,Z 1209.457,A -85,B 0,C 180,E1 380.475,E2 380.475} C_VEL
LIN {X 0,Y 87.181,Z 1204.504,A -85,B 0,C 180,E1 372.879,E2 372.879} C_VEL
LIN {X 0,Y 109.02,Z 1197.583,A -85,B 0,C 180,E1 367.905,E2 367.905} C_VEL
LIN {X 0,Y 129.439,Z 1189.657,A -85,B 0,C 180,E1 364.818,E2 364.818} C_VEL
LIN {X 0,Y 151.119,Z 1179.438,A -85,B 0,C 180,E1 362.473,E2 362.473} C_VEL
LIN {X 0,Y 151.736,Z 1179.122,A -85,B 0,C 180,E1 362.394,E2 362.394} C_VEL
LIN {X 0,Y 129.981,Z 1189.537,A -85,B 0,C 180,E1 359.978,E2 359.978} C_VEL
LIN {X 0,Y 108.177,Z 1198.148,A -85,B 0,C 180,E1 356.583,E2 356.583} C_VEL
LIN {X 0,Y 85.025,Z 1205.598,A -85,B 0,C 180,E1 351.043,E2 351.043} C_VEL
LIN {X 0,Y 64.021,Z 1210.977,A -85,B 0,C 180,E1 342.303,E2 342.303} C_VEL
LIN {X 0,Y 45.596,Z 1214.537,A -85,B 0,C 180,E1 326.437,E2 326.437} C_VEL
LIN {X 0,Y 34.228,Z 1216.447,A -85,B 0,C 180,E1 299.775,E2 299.775} C_VEL
LIN {X 0,Y 32.028,Z 1216.953,A -85,B 0,C 180,E1 271.789,E2 271.789} C_VEL
LIN {X 0,Y 32.507,Z 1216.711,A -85,B 0,C 180,E1 252.086,E2 252.086} C_VEL
LIN {X 0,Y 41.205,Z 1215.294,A -85,B 0,C 180,E1 220.447,E2 220.447} C_VEL
LIN {X 0,Y 45.466,Z 1214.402,A -85,B 0,C 180,E1 211.932,E2 211.932} C_VEL
LIN {X 0,Y 58.542,Z 1211.459,A -85,B 0,C 180,E1 192.692,E2 192.692} C_VEL
LIN {X 0,Y 63.641,Z 1210.316,A -85,B 0,C 180,E1 189.694,E2 189.694} C_VEL
LIN {X 0,Y 84.132,Z 1205.291,A -85,B 0,C 180,E1 183.357,E2 183.357} C_VEL
LIN {X 0,Y 108.435,Z 1197.638,A -85,B 0,C 180,E1 178.943,E2 178.943} C_VEL
LIN {X 0,Y 118.54,Z 1193.935,A -85,B 0,C 180,E1 177.583,E2 177.583} C_VEL
LIN {X 0,Y 96.439,Z 1201.499,A -85,B 0,C 180,E1 174.444,E2 174.444} C_VEL
LIN {X 0,Y 74.259,Z 1207.563,A -85,B 0,C 180,E1 169.388,E2 169.388} C_VEL
LIN {X 0,Y 53.059,Z 1211.777,A -85,B 0,C 180,E1 160.427,E2 160.427} C_VEL
LIN {X 0,Y 33.112,Z 1214.561,A -85,B 0,C 180,E1 139.018,E2 139.018} C_VEL
LIN {X 0,Y 24.776,Z 1215.383,A -85,B 0,C 180,E1 106.409,E2 106.409} C_VEL
LIN {X 0,Y 24.292,Z 1215.455,A -85,B 0,C 180,E1 80.524,E2 80.524} C_VEL
LIN {X 0,Y 31.18,Z 1214.782,A -85,B 0,C 180,E1 45.132,E2 45.132} C_VEL
LIN {X 0,Y 48.67,Z 1212.615,A -85,B 0,C 180,E1 22.413,E2 22.413} C_VEL
LIN {X 0,Y 69.518,Z 1208.657,A -85,B 0,C 180,E1 12.033,E2 12.033} C_VEL
LIN {X 0,Y 92.526,Z 1202.811,A -85,B 0,C 180,E1 6.187,E2 6.187} C_VEL
LIN {X 0,Y 113.137,Z 1196.056,A -85,B 0,C 180,E1 2.988,E2 2.988} C_VEL
LIN {X 0,Y 118.372,Z 1194.16,A -85,B 0,C 180,E1 2.342,E2 2.342} C_VEL
LIN {X 0,Y 95.999,Z 1201.9,A -85,B 0,C 180,E1 -0.934,E2 -0.934} C_VEL
LIN {X 0,Y 73.348,Z 1208.211,A -85,B 0,C 180,E1 -6.261,E2 -6.261} C_VEL
LIN {X 0,Y 52.821,Z 1212.49,A -85,B 0,C 180,E1 -15.12,E2 -15.12} C_VEL
LIN {X 0,Y 33.304,Z 1215.502,A -85,B 0,C 180,E1 -35.847,E2 -35.847} C_VEL
LIN {X 0,Y 24.495,Z 1216.567,A -85,B 0,C 180,E1 -70.94,E2 -70.94} C_VEL
LIN {X 0,Y 24.016,Z 1216.74,A -85,B 0,C 180,E1 -92.386,E2 -92.386} C_VEL
LIN {X 0,Y 27.943,Z 1216.141,A -85,B 0,C 180,E1 -130.097,E2 -130.097} C_VEL
LIN {X 0,Y 41.618,Z 1214.286,A -85,B 0,C 180,E1 -155.916,E2 -155.916} C_VEL
LIN {X 0,Y 62.007,Z 1210.688,A -85,B 0,C 180,E1 -169.613,E2 -169.613} C_VEL
LIN {X 0,Y 63.641,Z 1210.316,A -85,B 0,C 180,E1 -170.306,E2 -170.306} C_VEL
LIN {X 0,Y 67.859,Z 1209.321,A -85,B 0,C 180,E1 -172.857,E2 -172.857} C_VEL
LIN {X 0,Y 78.046,Z 1206.659,A -85,B 0,C 180,E1 -180.68,E2 -180.68} C_VEL
LIN {X 0,Y 82.035,Z 1205.602,A -85,B 0,C 180,E1 -181.965,E2 -181.965} C_VEL
LIN {X 0,Y 84.061,Z 1205.074,A -85,B 0,C 180,E1 -182.384,E2 -182.384} C_VEL
LIN {X 0,Y 62.45,Z 1209.996,A -85,B 0,C 180,E1 -186.952,E2 -186.952} C_VEL
LIN {X 0,Y 39.744,Z 1213.553,A -85,B 0,C 180,E1 -197.064,E2 -197.064} C_VEL
LIN {X 0,Y 21.812,Z 1215.35,A -85,B 0,C 180,E1 -222.823,E2 -222.823} C_VEL
LIN {X 0,Y 16.103,Z 1215.735,A -85,B 0,C 180,E1 -270,E2 -270} C_VEL
LIN {X 0,Y 23.151,Z 1215.247,A -85,B 0,C 180,E1 -321.021,E2 -321.021} C_VEL
LIN {X 0,Y 40.64,Z 1213.489,A -85,B 0,C 180,E1 -343.641,E2 -343.641} C_VEL
LIN {X 0,Y 63.411,Z 1209.875,A -85,B 0,C 180,E1 -353.399,E2 -353.399} C_VEL
LIN {X 0,Y 84.055,Z 1205.174,A -85,B 0,C 180,E1 -357.709,E2 -357.709} C_VEL
LIN {X 0,Y 62.047,Z 1210.337,A -85,B 0,C 180,E1 -362.44,E2 -362.44} C_VEL
LIN {X 0,Y 39.914,Z 1213.999,A -85,B 0,C 180,E1 -372.321,E2 -372.321} C_VEL
LIN {X 0,Y 22.333,Z 1215.958,A -85,B 0,C 180,E1 -396.306,E2 -396.306} C_VEL
LIN {X 0,Y 16.013,Z 1216.551,A -85,B 0,C 180,E1 -447.545,E2 -447.545} C_VEL
LIN {X 0,Y 18.714,Z 1216.243,A -85,B 0,C 180,E1 -489.878,E2 -489.878} C_VEL
LIN {X 0,Y 36.255,Z 1214.437,A -85,B 0,C 180,E1 -524.852,E2 -524.852} C_VEL
LIN {X 0,Y 57.13,Z 1211.215,A -85,B 0,C 180,E1 -536.018,E2 -536.018} C_VEL
LIN {X 0,Y 80.02,Z 1206.125,A -85,B 0,C 180,E1 -541.615,E2 -541.615} C_VEL
LIN {X 0,Y 82.035,Z 1205.602,A -85,B 0,C 180,E1 -541.965,E2 -541.965} C_VEL
LIN {X 0,Y 80.225,Z 1206.053,A -85,B 0,C 180,E1 -542.635,E2 -542.635} C_VEL
LIN {X 0,Y 70.307,Z 1208.395,A -85,B 0,C 180,E1 -543.113,E2 -543.113} C_VEL
LIN {X 0,Y 50.566,Z 1212.124,A -85,B 0,C 180,E1 -541.959,E2 -541.959} C_VEL
LIN {X 0,Y 36.282,Z 1214.073,A -85,B 0,C 180,E1 -538.511,E2 -538.511} C_VEL
LIN {X 0,Y 15.172,Z 1215.98,A -85,B 0,C 180,E1 -517.311,E2 -517.311} C_VEL
LIN {X 0,Y 8.008,Z 1216.351,A -85,B 0,C 180,E1 -447.231,E2 -447.231} C_VEL
LIN {X 0,Y 19.607,Z 1215.676,A -85,B 0,C 180,E1 -374.329,E2 -374.329} C_VEL
LIN {X 0,Y 38.995,Z 1213.789,A -85,B 0,C 180,E1 -360.416,E2 -360.416} C_VEL
LIN {X 0,Y 47.482,Z 1212.654,A -85,B 0,C 180,E1 -357.668,E2 -357.668} C_VEL
LIN {X 0,Y 24.658,Z 1215.066,A -85,B 0,C 180,E1 -346.699,E2 -346.699} C_VEL
LIN {X 0,Y 9.835,Z 1215.823,A -85,B 0,C 180,E1 -307.588,E2 -307.588} C_VEL
LIN {X 0,Y 8.893,Z 1215.855,A -85,B 0,C 180,E1 -243.272,E2 -243.272} C_VEL
LIN {X 0,Y 22.798,Z 1215.168,A -85,B 0,C 180,E1 -195.234,E2 -195.234} C_VEL
LIN {X 0,Y 45.058,Z 1212.971,A -85,B 0,C 180,E1 -183.075,E2 -183.075} C_VEL
LIN {X 0,Y 47.635,Z 1212.57,A -85,B 0,C 180,E1 -182.256,E2 -182.256} C_VEL
LIN {X 0,Y 36.282,Z 1214.073,A -85,B 0,C 180,E1 -178.511,E2 -178.511} C_VEL
LIN {X 0,Y 28.408,Z 1214.935,A -85,B 0,C 180,E1 -176.22,E2 -176.22} C_VEL
LIN {X 0,Y 15.146,Z 1215.811,A -85,B 0,C 180,E1 -176.72,E2 -176.72} C_VEL
LIN {X 0,Y 1.788,Z 1216.142,A -85,B 0,C 180,E1 -185.14,E2 -185.14} C_VEL
LIN {X 0,Y 0.547,Z 1216.141,A -85,B 0,C 180,E1 -352.717,E2 -352.717} C_VEL
LIN {X 0,Y 0.661,Z 1216.133,A -85,B 0,C 180,E1 -185.372,E2 -185.372} C_VEL
LIN {X 0,Y 0.547,Z 1216.141,A -85,B 0,C 180,E1 -352.717,E2 -352.717} C_VEL
LIN {X 0,Y 2.547,Z 1218.141,A -85,B 0,C 180,E1 -361.407,E2 -361.407} C_VEL
LIN {X 0,Y 2.547,Z 1240.5,A -85,B 0,C 180,E1 -361.407,E2 -361.407} C_VEL
LIN {X 0,Y 2.547,Z 1240.5,A -85,B 0,C 180,E1 -361.407,E2 -361.407}

QRS_NEXT_CUT()

QRS_NEXT()
QRS_HOME()

END
